I10:  NOP   0;
//
// copy state
      U     "G245M".Gr.InOutAutostartMan; // TRAVELLING DRIVE  GERM 8
      =     "MAL1S024Par".Ilo.GrSTMan[2];
      U     "G249M".Gr.InOutAutostartMan; // TURNING SCREWS  GERM 8
      =     "MAL1S024Par".Ilo.GrSTMan[6];
      U     "G250M".Gr.InOutAutostartMan; // FAN AND VALVE SRAY AIR  GERM 8
      =     "MAL1S024Par".Ilo.GrSTMan[7];
      U     "G251M".Gr.InOutAutostartMan; // FRESH AIR LOUVER  GERM 8
      =     "MAL1S024Par".Ilo.GrSTMan[8];
      U     "G257M".Gr.InOutAutostartMan; // COOLING / HEATING  GERM 8
      =     "MAL1S024Par".Ilo.GrSTMan[14];

// copy state

NETWORK
TITLE =ASW_9999: Init ASW Flags
// clear all flags explicde to find them back
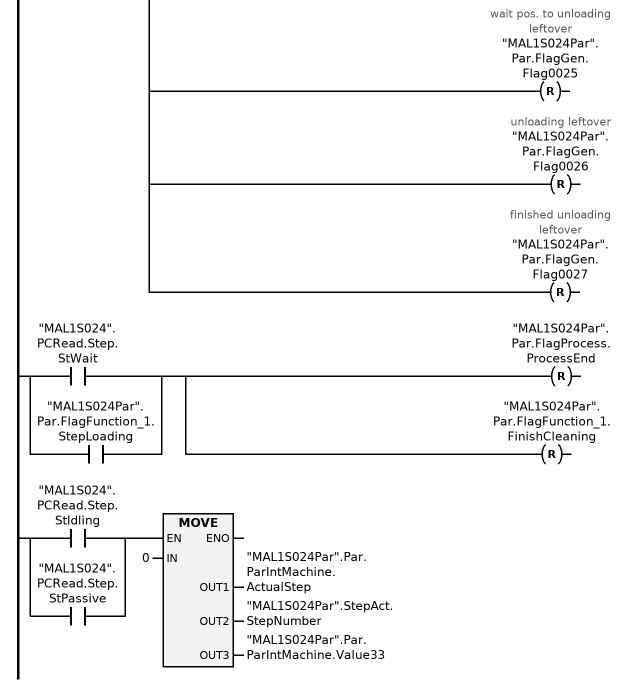
      U     "MAL1S024".PCRead.Step.StIdling;
      O     "MAL1S024".PCRead.Step.StPassive;
      R     "MAL1S024Par".Par.FlagFunction_1.StepLoading;
      R     "MAL1S024Par".Par.FlagFunction_1.StepUnloading;
      R     "MAL1S024Par".Par.FlagFunction_1.StepCleaning;
      R     "MAL1S024Par".Par.FlagFunction_1.LoadingBreak;
      R     "MAL1S024Par".Par.FlagFunction_1.UnloadingBreak;
      R     "MAL1S024Par".Par.FlagFunction_1.CleaningBreak;
      R     "MAL1S024Par".Par.FlagFunction_1.FinishLoading;
      R     "MAL1S024Par".Par.FlagFunction_1.FinishUnloading;
      R     "MAL1S024Par".Par.FlagFunction_1.FinishCleaning;
      R     "MAL1S024Par".Par.FlagFunction_1.Round_1;
      R     "MAL1S024Par".Par.FlagFunction_1.Round_2;
      R     "MAL1S024Par".Par.FlagFunction_1.Round_3;
      R     "MAL1S024Par".Par.FlagFunction_1.Round_4;
      R     "MAL1S024Par".Par.FlagFunction_1.Round_5;
      R     "MAL1S024Par".Par.FlagFunction_1.Round_6;
      R     "MAL1S024Par".Par.FlagFunction_1.Beladung_beendet;
      R     "MAL1S024Par".Par.FlagFunction_1.Entladerunden_erreicht;
      R     "MAL1S024Par".Par.FlagFunction_1.Reinigungsrunde_erreicht;
      R     "MAL1S024Par".Par.FlagGen.TurningStarted;
      R     "MAL1S024Par".Par.FlagFunction_1.TurningStart;
      R     "MAL1S024Par".Par.FlagFunction_1.TurningStop;
      R     "MAL1S024Par".Par.FlagFunction_1.TurningLeft;
      R     "MAL1S024Par".Par.FlagFunction_1.TurningRight;
      R     "MAL1S024Par".Par.FlagFunction_1.LoadFirstPartEnd;
      R     "MAL1S024Par".Par.FlagFunction_1.TurningWithSpraying;
      R     "MAL1S024Par".Par.FlagFunction_1.TurningWithoutSpraying;
      R     "MAL1S024Par".Par.FlagGen.TurningStarted;
      R     "MAL1S024Par".Par.FlagProcess2.Turning1WithoutSpraying;
      R     "MAL1S024Par".Par.FlagProcess2.Turning2WithoutSpraying;
      R     "MAL1S024Par".Par.FlagProcess2.Turning1WithSpraying;
      R     "MAL1S024Par".Par.FlagProcess2.Turning2WithSpraying;
      R     "MAL1S024Par".Par.FlagProcess2.Turning1WithDosing;
      R     "MAL1S024Par".Par.FlagProcess2.Turning2WithDosing;
      R     "MAL1S024Par".Par.FlagProcess2.StartFirstTurningRound;
      R     "MAL1S024Par".Par.FlagProcess2.StartSecondTurningRound;

      R     "MAL1S024Par".Par.FlagFunction_1.UnloadFirstPartEnd;
      R     "MAL1S024Par".Par.FlagFunction_1.UnloadSecondPartEnd;
      R     "MAL1S024Par".Par.FlagFunction_1.UnloadFirstPart;
      R     "MAL1S024Par".Par.FlagFunction_1.UnloadSecondPart;
      R     "MAL1S024Par".Par.FlagFunction_1.UnloadingStarted;
      R     "MAL1S024Par".Par.FlagProcess.ProcessActive;
      R     "MAL1S024Par".Par.FlagProcess.ProcessStartFP;
      R     "MAL1S024Par".Par.FlagProcess.ProcessStartScan;
      R     "MAL1S024Par".Par.FlagProcess.ProcessEnd;
      R     "MAL1S024Par".Par.FlagProcess.FP_SendResultToPIC;
      R     "MAL1S024Par".Par.FlagMachine.ImpulsNullstellung;
      R     "MAL1S024Par".Par.FlagMachine_0.CmdTurnRevAfterUnloading;
      R     "MAL1S024Par".Par.FlagMachine_0.CleaningAfterUnloading;
      R     "MAL1S024Par".Par.FlagMachine_0.CleaningAfterLoading;

      R     "MAL1S024Par".Par.FlagGen.Flag0024; // finished first unloading
      R     "MAL1S024Par".Par.FlagGen.Flag0025; // wait pos. to unloading leftover
      R     "MAL1S024Par".Par.FlagGen.Flag0026; // unloading leftover
      R     "MAL1S024Par".Par.FlagGen.Flag0027; // finished unloading leftover

//
      U     "MAL1S024".PCRead.Step.StWait;
      O     "MAL1S024Par".Par.FlagFunction_1.StepLoading;
      R     "MAL1S024Par".Par.FlagProcess.ProcessEnd;
      R     "MAL1S024Par".Par.FlagFunction_1.FinishCleaning;

      U     "MAL1S024".PCRead.Step.StIdling;
      O     "MAL1S024".PCRead.Step.StPassive;
      SPBN  csn;
      L     0; // clear step number
      T     "MAL1S024Par".Par.ParIntMachine.ActualStep;
      T     "MAL1S024Par".StepAct.StepNumber;
      T     "MAL1S024Par".Par.ParIntMachine.Value33; //aktuelle Wartezeit Maschine bei 100% Unloading-Position
csn:  NOP   0;

NETWORK
TITLE =Main0_End: Init flag
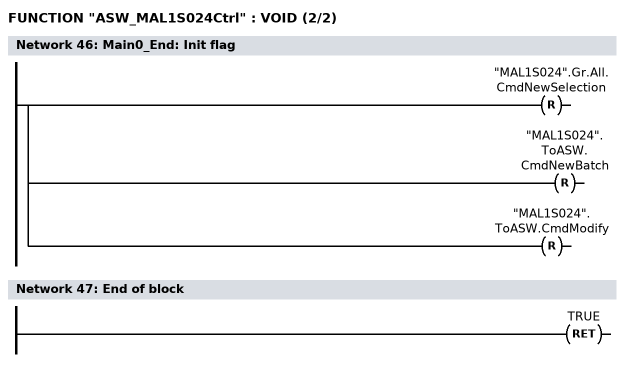

      SET   ;
      R     "MAL1S024".Gr.All.CmdNewSelection;
      R     "MAL1S024".ToASW.CmdNewBatch;
      R     "MAL1S024".ToASW.CmdModify;

NETWORK
TITLE =End of block

      BE    ;

END_FUNCTION

